SUBAPPLICATION mapping_Uebung_033 (* LED Strip Blinkende LED *)
  (* Standard: 61499-2 *)
  (* Version 1.0, 2023-10-23, franz *)
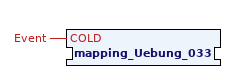
  EVENT_INPUT
    COLD;
  END_EVENT
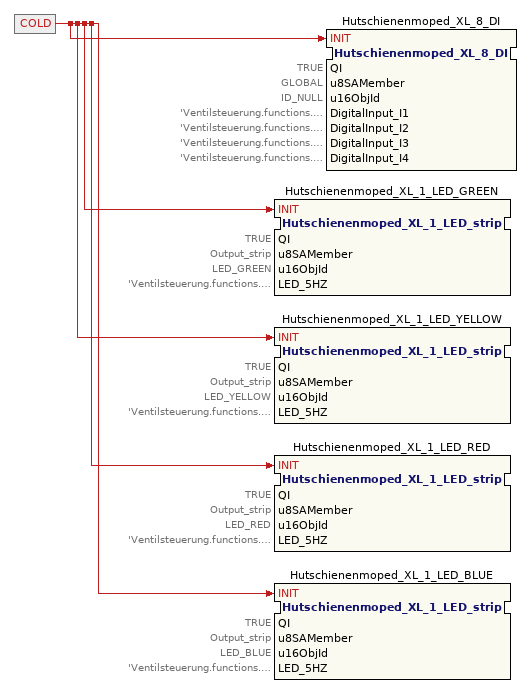
  FBS
    Hutschienenmoped_XL_8_DI : Hutschienenmoped_XL_8_DI(QI := TRUE, u8SAMember := GLOBAL, u16ObjId := ID_NULL, DigitalInput_I1 := 'Ventilsteuerung.functions.BUTTON_GREEN', DigitalInput_I2 := 'Ventilsteuerung.functions.BUTTON_YELLOW', DigitalInput_I3 := 'Ventilsteuerung.functions.BUTTON_RED', DigitalInput_I4 := 'Ventilsteuerung.functions.BUTTON_BLUE');
    Hutschienenmoped_XL_1_LED_YELLOW : Hutschienenmoped_XL_1_LED_strip(QI := TRUE, u8SAMember := Output_strip, u16ObjId := LED_YELLOW, LED_5HZ := 'Ventilsteuerung.functions.LED_YELLOW_5HZ');
    Hutschienenmoped_XL_1_LED_GREEN : Hutschienenmoped_XL_1_LED_strip(QI := TRUE, u8SAMember := Output_strip, u16ObjId := LED_GREEN, LED_5HZ := 'Ventilsteuerung.functions.LED_GREEN_5HZ');
    Hutschienenmoped_XL_1_LED_RED : Hutschienenmoped_XL_1_LED_strip(QI := TRUE, u8SAMember := Output_strip, u16ObjId := LED_RED, LED_5HZ := 'Ventilsteuerung.functions.LED_RED_5HZ');
    Hutschienenmoped_XL_1_LED_BLUE : Hutschienenmoped_XL_1_LED_strip(QI := TRUE, u8SAMember := Output_strip, u16ObjId := LED_BLUE, LED_5HZ := 'Ventilsteuerung.functions.LED_BLUE_5HZ');
  END_FBS
  EVENT_CONNECTIONS
    COLD TO Hutschienenmoped_XL_8_DI.INIT;
    COLD TO Hutschienenmoped_XL_1_LED_YELLOW.INIT;
    COLD TO Hutschienenmoped_XL_1_LED_GREEN.INIT;
    COLD TO Hutschienenmoped_XL_1_LED_RED.INIT;
    COLD TO Hutschienenmoped_XL_1_LED_BLUE.INIT;
  END_CONNECTIONS
END_SUBAPPLICATION
